TYPE ST_GearAxis_back :
STRUCT
    index   :   UINT:=1;    //index of master axis
    ratio   :   LREAL;      //gearing ratio
END_STRUCT
END_TYPE

(* stored: Version 1.1.0.1, ProductVersion 3.1.4024.6
   DUT ST_GearAxis_back: Id {265c814e-8429-46d8-bc92-5fd53f51700c} *)
